FUNCTION_BLOCK NormallyClosedPushButton IMPLEMENTS I_PushButton
VAR
	input AT %I*	:	BOOL;
END_VAR

PROPERTY PUBLIC IsPressed : BOOL

// ho eliminato manualmente il Setter di questa proprietà perché qui non ha senso
GET
IsPressed := NOT input;
END_GET
END_PROPERTY

PROPERTY PUBLIC IsReleased : BOOL

// ho eliminato manualmente il Setter di questa proprietà perché qui non ha senso
GET
IsReleased := NOT IsPressed;
END_GET
END_PROPERTY

END_FUNCTION_BLOCK

(* stored: Version 1.1.0.1, ProductVersion 3.1.4024.11
   POU NormallyClosedPushButton: Id {dc763925-e444-42e7-806d-7e2661aae3ae}, SpecialFunc None
   Property IsPressed: Id {10c582a4-a9eb-496d-9eba-e553c86703ea}
   Get Get: Id {62e67e1c-fb7e-4ef9-b8da-52a8692b14f7}
   Property IsReleased: Id {9b823a2c-121e-4821-96ff-d7e27f7c7e5a}
   Get Get: Id {c0c697fd-6b2b-4c66-a436-bd43201ded03} *)
